INTERFACE ITF_GroupE_TE1 EXTENDS ITF_BaseGroupElement

METHOD testMethodGE : BOOL
VAR_INPUT
END_VAR
END_METHOD

END_INTERFACE

(* stored: Version 1.1.0.1, ProductVersion 3.1.4024.15
   Itf ITF_GroupE_TE1: Id {8c2e7460-d2fc-4270-8aad-d79cbefea607}
   Method testMethodGE: Id {8dfc04b0-1810-4a33-a7fd-9741a961ad79} *)
